// TIA Portal V17 export
// export: Created 2025-03-07T09:24:37.7022115Z, ExportSetting WithDefaults, DisplayName Totally Integrated Automation Portal, DisplayVersion V17 Update 8, DisplayName TIA Portal Openness, DisplayVersion V17 Update 8, DisplayName TIA Portal Version Control Interface, DisplayVersion V17, DisplayName SINAMICS Startdrive Advanced, DisplayVersion V17 SP2, DisplayName SINAMICS Startdrive G110M, G120, G120C, G120D, G120P, G115D, DisplayVersion V17 SP2, DisplayName SINAMICS Startdrive G130, G150, S120, S150, SINAMICS MV, S210, DisplayVersion V17 SP2, DisplayName STEP 7 Professional, DisplayVersion V17 Update 8, DisplayName SINUMERIK ONE STEP 7 Toolbox, DisplayVersion V17 Update 12, DisplayName SINUMERIK 840D sl STEP 7 Toolbox, DisplayVersion V17 Update 12, DisplayName STEP 7 Safety, DisplayVersion V17 Update 6, DisplayName WinCC Advanced, DisplayVersion V17 Update 8
TYPE "MOTOR_CONTROL_DATA"
// stored: IsFailsafeCompliant false
   STRUCT
      Start : Bool;
      Conditions : Bool;
      CCW_Rotation : Bool;
      CW_Rotation : Bool;
      "Manual Speed" : Real;
      "Consignment Speed" : Real;
      Min_Range : Real;
      Max_Range : Real;
      Lim_Lo : Real;
      Lim_HI : Real;
      Analog_Lo : Real;
      Analog_Hi : Real;
      "HMI Manual Cons." : Real;
      "HMI Consignment" : Real;
      "HMI Feedback Value" : Real;
   END_STRUCT;
END_TYPE
